% RSLogix 500 project PLC_1_L3_3.RSS, saved by version 12.00.00.00 %
PROJECT "UNTITLED"    % processor: Bul.1763 MicroLogix 1100 Series B %

PROGRAM FILES
  LAD 2   2 rungs

DATA FILES
  O0 OUTPUT  5 elements
  I1 INPUT  6 elements
  S2 STATUS  66 elements
  B3 BINARY  1 elements
  T4 TIMER  1 elements
  C5 COUNTER  1 elements
  R6 CONTROL  1 elements
  N7 INTEGER  100 elements
  F8 FLOAT  1 elements
  B9 NBDF  10 elements  % New Binary Data File %
  N10 NIDF  10 elements  % New Integer Data File %

LADDER 2
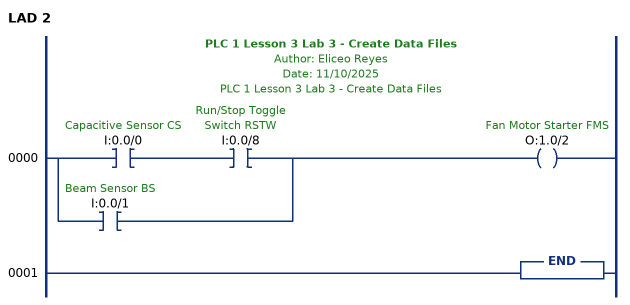
% Rung: 0 %
% TITLE: PLC 1 Lesson 3 Lab 3 - Create Data Files %
% Author: Eliceo Reyes
% Date: 11/10/2025
% PLC 1 Lesson 3 Lab 3 - Create Data Files %
SOR BST XIC I:0.0/0 XIC I:0.0/8 NXB XIC I:0.0/1 BND OTE O:1.0/2 EOR
%   I:0.0/0  CS  "Capacitive Sensor" %
%   I:0.0/8  RSTW  "Run/Stop Toggle Switch" %
%   I:0.0/1  BS  "Beam Sensor" %
%   O:1.0/2  FMS  "Fan Motor Starter" %
% Rung: 1 %
SOR END EOR
